FUNCTION_BLOCK PoolDeleteVersion (* Service Interface Block to delete a stored object pool version from VT flash *)
  (* Standard: ISO 11783-6; Description: Copyright (c) 2025 Meisterschulen am Ostbahnhof This program and the accompanying materials are made available under the terms of the Eclipse Public License 2.0 which is available at https://www.eclipse.org/legal/epl-2.0/ SPDX-License-Identifier: EPL-2.0 Service Interface Block to delete a stored object pool version from VT flash This block wraps the functionality of VTC_PoolDeleteVersion() from the ISOBUS driver samples. It allows deleting a stored object pool version from the VT's non-volatile memory. The block calls IsoVtcCmd_DeleteVersion() to remove the specified pool version. Parameters: - versionString: The version label of the pool to delete (max 32 bytes, zero-terminated) Use spaces ( '      ' ) to delete the last stored pool from flash - u8Instance: The VT client instance identifier Typical use cases: - Delete old pool versions before uploading a new one - Clean up flash memory on the VT - Remove corrupted pool versions Note: The version string must be zero-terminated or exactly 32 bytes long (ISO V11+). *)
  (* Version 1.0, 2025-02-27, Generated, Meisterschulen am Ostbahnhof, initial API and implementation and/or initial documentation *)
  PACKAGE isobus::UT::util;
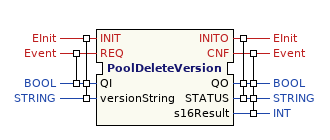
  EVENT_INPUT
    INIT : EInit WITH QI, versionString; (* Service Initialization *)
    REQ WITH QI; (* Service Request - Delete pool version *)
  END_EVENT
  EVENT_OUTPUT
    INITO : EInit WITH QO, STATUS; (* Initialization Confirm *)
    CNF WITH QO, STATUS, s16Result; (* Confirmation - Pool deletion completed *)
  END_EVENT
  VAR_INPUT
    QI : BOOL; (* Quality Input - TRUE to enable service *)
    versionString : STRING := '       '; (* Version label to delete (use spaces for last stored pool) *)
  END_VAR
  VAR_OUTPUT
    QO : BOOL; (* Quality Output - TRUE if deletion was successful *)
    STATUS : STRING; (* Service Status *)
    s16Result : INT; (* Return value: 0=E_NO_ERR (success), negative=error code *)
  END_VAR
END_FUNCTION_BLOCK
